FUNCTION_BLOCK FB_Janitza
VAR_IN_OUT
	get					: ST_PowerMonitor_get;
END_VAR
VAR
	MBRead: FB_MBReadRegs;
	w_MBStartAddress	:	WORD;
	//Set 1 is bigger, as this includes voltage measurements.
	DataBuffer		: 	ARRAY[0..62] OF REAL;
	SecondDataBuffer		: 	ARRAY[0..62] OF REAL;
	tempword	:	dword;	
	temp	:	BOOL;
	UI_Iterator	:	UINT;
	//retrieve new data every 100ms
	GetDataTimer	:	TON := (PT := TIME#100MS);
END_VAR

VAR_INPUT
	ReadData: BOOL;
	b_TNmodeEnable		AT %Q* : BOOL;
END_VAR

VAR
	ast_InputPowerlockData	:	ARRAY[1..2] OF ST_Powerlockdata;
	ast_OutputPowerlockData	:	ARRAY[1..3] OF ST_Powerlockdata;

	StartTransmissionEdge : R_Trig;
	TransmissionDone	:	F_trig;
	
	ui_MBRetryCount	:	uint;
	
	b_busy: BOOL;
	b_CommError: BOOL;
	udi_errid: UDINT;
	udi_cbread: UDINT;
	
	testWord	:	DWORD;
	testWordB	:	WORD;
	testWordC	:	WORD;
END_VAR



//While ReadData is true, initiate data transfer every 100ms;
GetDataTimer(in:= ((NOT GetDataTimer.Q) AND ReadData));

//ReadJanitzaData();
ReadDataSFC();

ACTION aCombineInputData:
IF PowerMeterConfig.b_InputFieldsAvailable THEN
	//Combine shared data from output fields into get struct
	get.InputField.r_Current[Phases.L1] :=	get.InputField.ar_PowerlockCurrents[1][Phases.L1] + 
											get.InputField.ar_PowerlockCurrents[2][Phases.L1];
	
	get.InputField.r_Current[Phases.L2] :=	get.InputField.ar_PowerlockCurrents[1][Phases.L2] + 
											get.InputField.ar_PowerlockCurrents[2][Phases.L2];
	
	get.InputField.r_Current[Phases.L3] :=	get.InputField.ar_PowerlockCurrents[1][Phases.L3] + 
											get.InputField.ar_PowerlockCurrents[2][Phases.L3];			
	
	get.InputField.r_Current[Phases.N] :=	get.InputField.ar_PowerlockCurrents[1][Phases.N] + 
											get.InputField.ar_PowerlockCurrents[2][Phases.N];			
	
	get.InputField.r_Current[Phases.AVG] :=	(get.InputField.r_Current[Phases.L1] + 
											get.InputField.r_Current[Phases.L2] +
											get.InputField.r_Current[Phases.L3])/3;							
	
	Get.InputField.r_ActivePhasePower[Phases.L1]	:=	ast_InputPowerLockData[1].r_ActivePhasePower[Phases.L1] + 
														ast_InputPowerLockData[2].r_ActivePhasePower[Phases.L1];
	
	Get.InputField.r_ActivePhasePower[Phases.L2]	:=	ast_InputPowerLockData[1].r_ActivePhasePower[Phases.L2] + 
														ast_InputPowerLockData[2].r_ActivePhasePower[Phases.L2];
														
	Get.InputField.r_ActivePhasePower[Phases.L3]	:=	ast_InputPowerLockData[1].r_ActivePhasePower[Phases.L3] + 
														ast_InputPowerLockData[2].r_ActivePhasePower[Phases.L3];
														
	Get.InputField.r_ActivePhasePower[Phases.AVG]	:=	ast_InputPowerLockData[1].r_ActivePhasePower[Phases.AVG] + 
														ast_InputPowerLockData[2].r_ActivePhasePower[Phases.AVG];									
	
														
														
	Get.InputField.r_ApparentPhasePower[Phases.L1]	:=	ast_InputPowerLockData[1].r_ApparentPhasePower[Phases.L1] + 
														ast_InputPowerLockData[2].r_ApparentPhasePower[Phases.L1];
	
	Get.InputField.r_ApparentPhasePower[Phases.L2]	:=	ast_InputPowerLockData[1].r_ApparentPhasePower[Phases.L2] + 
														ast_InputPowerLockData[2].r_ApparentPhasePower[Phases.L2];
														
	Get.InputField.r_ApparentPhasePower[Phases.L3]	:=	ast_InputPowerLockData[1].r_ApparentPhasePower[Phases.L3] + 
														ast_InputPowerLockData[2].r_ApparentPhasePower[Phases.L3];
														
	Get.InputField.r_ApparentPhasePower[Phases.AVG]	:=	ast_InputPowerLockData[1].r_ApparentPhasePower[Phases.AVG] + 
														ast_InputPowerLockData[2].r_ApparentPhasePower[Phases.AVG];	

														
														
	Get.InputField.r_ReactivePhasePower[Phases.L1]	:=	ast_InputPowerLockData[1].r_ReactivePhasePower[Phases.L1] + 
														ast_InputPowerLockData[2].r_ReactivePhasePower[Phases.L1];
	
	Get.InputField.r_ReactivePhasePower[Phases.L2]	:=	ast_InputPowerLockData[1].r_ReactivePhasePower[Phases.L2] + 
														ast_InputPowerLockData[2].r_ReactivePhasePower[Phases.L2];
														
	Get.InputField.r_ReactivePhasePower[Phases.L3]	:=	ast_InputPowerLockData[1].r_ReactivePhasePower[Phases.L3] + 
														ast_InputPowerLockData[2].r_ReactivePhasePower[Phases.L3];
														
	Get.InputField.r_ReactivePhasePower[Phases.AVG]	:=	ast_InputPowerLockData[1].r_ReactivePhasePower[Phases.AVG] + 
														ast_InputPowerLockData[2].r_ReactivePhasePower[Phases.AVG];	


										
	Get.InputField.r_ActivePower		:=	ast_InputPowerLockData[1].r_ActivePower + 
											ast_InputPowerLockData[2].r_ActivePower;
	
	Get.InputField.r_ApparentPower		:=	ast_InputPowerLockData[1].r_ApparentPower + 
											ast_InputPowerLockData[2].r_ApparentPower;
											
	Get.InputField.r_ReactivePower		:=	ast_InputPowerLockData[1].r_ReactivePower + 
											ast_InputPowerLockData[2].r_ReactivePower;
	
	Get.InputField.r_EnergyConsumed		:=	ast_InputPowerLockData[1].r_EnergyConsumed + 
											ast_InputPowerLockData[2].r_EnergyConsumed;
	
	Get.InputField.r_EnergySupplied		:=	ast_InputPowerLockData[1].r_EnergySupplied + 
											ast_InputPowerLockData[2].r_EnergySupplied;
	
	get.InputField.r_PowerFactor[Phases.L1] :=		(ast_InputPowerLockData[1].ar_PowerFactor[Phases.L1] + 
													ast_InputPowerLockData[2].ar_PowerFactor[Phases.L1] )/2;	
														
	get.InputField.r_PowerFactor[Phases.L2] :=		(ast_InputPowerLockData[1].ar_PowerFactor[Phases.L2] + 
													ast_InputPowerLockData[2].ar_PowerFactor[Phases.L2])/2;		
	
	get.InputField.r_PowerFactor[Phases.L3] :=		(ast_InputPowerLockData[1].ar_PowerFactor[Phases.L3] + 
													ast_InputPowerLockData[2].ar_PowerFactor[Phases.L3])/2;
	
	get.InputField.r_THD[Phases.L1] 		:=		(ast_InputPowerLockData[1].ar_THD[Phases.L1] + 
													ast_InputPowerLockData[2].ar_THD[Phases.L1])/2;
														
	get.InputField.r_THD[Phases.L2] 		:=		(ast_InputPowerLockData[1].ar_THD[Phases.L2] + 
													ast_InputPowerLockData[2].ar_THD[Phases.L2])/2;	
	
	get.InputField.r_THD[Phases.L3]		 	:=		(ast_InputPowerLockData[1].ar_THD[Phases.L3] + 
													ast_InputPowerLockData[2].ar_THD[Phases.L3])/2;											
	
	get.InputField.r_PowerFactor[Phases.AVG] :=	(get.InputField.r_PowerFactor[Phases.L1] + 
													get.InputField.r_PowerFactor[Phases.L2] + 
													get.InputField.r_PowerFactor[Phases.L3])/3;		
	
	get.InputField.r_THD[Phases.AVG] :=			(get.InputField.r_THD[Phases.L1] + 
													get.InputField.r_THD[Phases.L2] + 
													get.InputField.r_THD[Phases.L3])/3;
end_if
END_ACTION

ACTION aCombineOutputData:

//Combine shared data from output fields into get struct
get.OutputField.r_Current[Phases.L1] :=	get.OutputField.ar_PowerlockCurrents[1][Phases.L1] + 
										get.OutputField.ar_PowerlockCurrents[2][Phases.L1] + 
										get.OutputField.ar_PowerlockCurrents[3][Phases.L1];

get.OutputField.r_Current[Phases.L2] :=	get.OutputField.ar_PowerlockCurrents[1][Phases.L2] + 
										get.OutputField.ar_PowerlockCurrents[2][Phases.L2] + 
										get.OutputField.ar_PowerlockCurrents[3][Phases.L2];

get.OutputField.r_Current[Phases.L3] :=	get.OutputField.ar_PowerlockCurrents[1][Phases.L3] + 
										get.OutputField.ar_PowerlockCurrents[2][Phases.L3] + 
										get.OutputField.ar_PowerlockCurrents[3][Phases.L3];			

get.OutputField.r_Current[Phases.N] :=	get.OutputField.ar_PowerlockCurrents[1][Phases.N] + 
										get.OutputField.ar_PowerlockCurrents[2][Phases.N] + 
										get.OutputField.ar_PowerlockCurrents[3][Phases.N];			

get.OutputField.r_Current[Phases.AVG] :=	(get.OutputField.r_Current[Phases.L1] + 
											get.OutputField.r_Current[Phases.L2] +
											get.OutputField.r_Current[Phases.L3])/3;							

Get.OutputField.r_ActivePhasePower[Phases.L1]	:=	ast_OutputPowerLockData[1].r_ActivePhasePower[Phases.L1] + 
													ast_OutputPowerLockData[2].r_ActivePhasePower[Phases.L1] +
													ast_OutputPowerLockData[3].r_ActivePhasePower[Phases.L1];
	
Get.OutputField.r_ActivePhasePower[Phases.L2]	:=	ast_OutputPowerLockData[1].r_ActivePhasePower[Phases.L2] + 
													ast_OutputPowerLockData[2].r_ActivePhasePower[Phases.L2] +
													ast_OutputPowerLockData[3].r_ActivePhasePower[Phases.L2];
														
Get.OutputField.r_ActivePhasePower[Phases.L3]	:=	ast_OutputPowerLockData[1].r_ActivePhasePower[Phases.L3] + 
													ast_OutputPowerLockData[2].r_ActivePhasePower[Phases.L3] + 
													ast_OutputPowerLockData[3].r_ActivePhasePower[Phases.L3];
														
Get.OutputField.r_ActivePhasePower[Phases.AVG]	:=	ast_OutputPowerLockData[1].r_ActivePhasePower[Phases.AVG] + 
													ast_OutputPowerLockData[2].r_ActivePhasePower[Phases.AVG] +
													ast_OutputPowerLockData[3].r_ActivePhasePower[Phases.AVG];									
	
														
														
Get.OutputField.r_ApparentPhasePower[Phases.L1]	:=	ast_OutputPowerLockData[1].r_ApparentPhasePower[Phases.L1] + 
													ast_OutputPowerLockData[2].r_ApparentPhasePower[Phases.L1] +
													ast_OutputPowerLockData[3].r_ApparentPhasePower[Phases.L1];
	
Get.OutputField.r_ApparentPhasePower[Phases.L2]	:=	ast_OutputPowerLockData[1].r_ApparentPhasePower[Phases.L2] + 
													ast_OutputPowerLockData[2].r_ApparentPhasePower[Phases.L2] +
													ast_OutputPowerLockData[3].r_ApparentPhasePower[Phases.L2];
														
Get.OutputField.r_ApparentPhasePower[Phases.L3]	:=	ast_OutputPowerLockData[1].r_ApparentPhasePower[Phases.L3] + 
													ast_OutputPowerLockData[2].r_ApparentPhasePower[Phases.L3] +
													ast_OutputPowerLockData[3].r_ApparentPhasePower[Phases.L3];
														
Get.OutputField.r_ApparentPhasePower[Phases.AVG]:=	ast_OutputPowerLockData[1].r_ApparentPhasePower[Phases.AVG] + 
													ast_OutputPowerLockData[2].r_ApparentPhasePower[Phases.AVG] +
													ast_OutputPowerLockData[3].r_ApparentPhasePower[Phases.AVG];	
														
													
													
Get.OutputField.r_ReactivePhasePower[Phases.L1]	:=	ast_OutputPowerLockData[1].r_ReactivePhasePower[Phases.L1] + 
													ast_OutputPowerLockData[2].r_ReactivePhasePower[Phases.L1] +
													ast_OutputPowerLockData[3].r_ReactivePhasePower[Phases.L1];	
	
Get.OutputField.r_ReactivePhasePower[Phases.L2]	:=	ast_OutputPowerLockData[1].r_ReactivePhasePower[Phases.L2] + 
													ast_OutputPowerLockData[2].r_ReactivePhasePower[Phases.L2] +
													ast_OutputPowerLockData[3].r_ReactivePhasePower[Phases.L2];	
														
Get.OutputField.r_ReactivePhasePower[Phases.L3]	:=	ast_OutputPowerLockData[1].r_ReactivePhasePower[Phases.L3] + 
													ast_OutputPowerLockData[2].r_ReactivePhasePower[Phases.L3] +
													ast_OutputPowerLockData[3].r_ReactivePhasePower[Phases.L3];	
														
Get.OutputField.r_ReactivePhasePower[Phases.AVG]:=	ast_OutputPowerLockData[1].r_ReactivePhasePower[Phases.AVG] + 
													ast_OutputPowerLockData[2].r_ReactivePhasePower[Phases.AVG] +	
													ast_OutputPowerLockData[3].r_ReactivePhasePower[Phases.AVG];												
											
											
Get.OutputField.r_ActivePower		:=	ast_OutputPowerLockData[1].r_ActivePower + 
										ast_OutputPowerLockData[2].r_ActivePower + 
										ast_OutputPowerLockData[3].r_ActivePower;

Get.OutputField.r_ApparentPower		:=	ast_OutputPowerLockData[1].r_ApparentPower + 
										ast_OutputPowerLockData[2].r_ApparentPower + 
										ast_OutputPowerLockData[3].r_ApparentPower;

Get.OutputField.r_ReactivePower		:=	ast_OutputPowerLockData[1].r_ReactivePower + 
										ast_OutputPowerLockData[2].r_ReactivePower + 
										ast_OutputPowerLockData[3].r_ReactivePower;

Get.OutputField.r_EnergyConsumed	:=	ast_OutputPowerLockData[1].r_EnergyConsumed + 
										ast_OutputPowerLockData[2].r_EnergyConsumed + 
										ast_OutputPowerLockData[3].r_EnergyConsumed;

Get.OutputField.r_EnergySupplied	:=	ast_OutputPowerLockData[1].r_EnergySupplied + 
										ast_OutputPowerLockData[2].r_EnergySupplied + 
										ast_OutputPowerLockData[3].r_EnergySupplied;

//if 3 output fields are available, calculate averages over 3 fields. Otherwise over 2
IF PowerMeterConfig.b_ThirdOutputFieldAvailable THEN
	get.OutputField.r_PowerFactor[Phases.L1] :=		(ast_OutputPowerLockData[1].ar_PowerFactor[Phases.L1] + 
													ast_OutputPowerLockData[2].ar_PowerFactor[Phases.L1] + 
													ast_OutputPowerLockData[3].ar_PowerFactor[Phases.L1])/3;	
													
	get.OutputField.r_PowerFactor[Phases.L2] :=		(ast_OutputPowerLockData[1].ar_PowerFactor[Phases.L2] + 
													ast_OutputPowerLockData[2].ar_PowerFactor[Phases.L2] + 
													ast_OutputPowerLockData[3].ar_PowerFactor[Phases.L2])/3;		

	get.OutputField.r_PowerFactor[Phases.L3] :=		(ast_OutputPowerLockData[1].ar_PowerFactor[Phases.L3] + 
													ast_OutputPowerLockData[2].ar_PowerFactor[Phases.L3] + 
													ast_OutputPowerLockData[3].ar_PowerFactor[Phases.L3])/3;	

	get.OutputField.r_THD[Phases.L1] 		:=		(ast_OutputPowerLockData[1].ar_THD[Phases.L1] + 
													ast_OutputPowerLockData[2].ar_THD[Phases.L1] + 
													ast_OutputPowerLockData[3].ar_THD[Phases.L1])/3;	
													
	get.OutputField.r_THD[Phases.L2] 		:=		(ast_OutputPowerLockData[1].ar_THD[Phases.L2] + 
													ast_OutputPowerLockData[2].ar_THD[Phases.L2] + 
													ast_OutputPowerLockData[3].ar_THD[Phases.L2])/3;		

	get.OutputField.r_THD[Phases.L3]		 :=		(ast_OutputPowerLockData[1].ar_THD[Phases.L3] + 
													ast_OutputPowerLockData[2].ar_THD[Phases.L3] + 
													ast_OutputPowerLockData[3].ar_THD[Phases.L3])/3;														
ELSE
	get.OutputField.r_PowerFactor[Phases.L1] :=		(ast_OutputPowerLockData[1].ar_PowerFactor[Phases.L1] + 
													ast_OutputPowerLockData[2].ar_PowerFactor[Phases.L1] )/2;	
													
	get.OutputField.r_PowerFactor[Phases.L2] :=		(ast_OutputPowerLockData[1].ar_PowerFactor[Phases.L2] + 
													ast_OutputPowerLockData[2].ar_PowerFactor[Phases.L2])/2;		

	get.OutputField.r_PowerFactor[Phases.L3] :=		(ast_OutputPowerLockData[1].ar_PowerFactor[Phases.L3] + 
													ast_OutputPowerLockData[2].ar_PowerFactor[Phases.L3])/2;

	get.OutputField.r_THD[Phases.L1] 		:=		(ast_OutputPowerLockData[1].ar_THD[Phases.L1] + 
													ast_OutputPowerLockData[2].ar_THD[Phases.L1])/2;
													
	get.OutputField.r_THD[Phases.L2] 		:=		(ast_OutputPowerLockData[1].ar_THD[Phases.L2] + 
													ast_OutputPowerLockData[2].ar_THD[Phases.L2])/2;	

	get.OutputField.r_THD[Phases.L3]		 :=		(ast_OutputPowerLockData[1].ar_THD[Phases.L3] + 
													ast_OutputPowerLockData[2].ar_THD[Phases.L3])/2;											
END_IF



get.OutputField.r_PowerFactor[Phases.AVG] :=	(get.OutputField.r_PowerFactor[Phases.L1] + 
												get.OutputField.r_PowerFactor[Phases.L2] + 
												get.OutputField.r_PowerFactor[Phases.L3])/3;		

get.OutputField.r_THD[Phases.AVG] :=			(get.OutputField.r_THD[Phases.L1] + 
												get.OutputField.r_THD[Phases.L2] + 
												get.OutputField.r_THD[Phases.L3])/3;
END_ACTION

ACTION aReadInputField1:

IF NOT PowerMeterConfig.b_InputFieldsAvailable THEN
	//skip this step if input fields are not in use
	SFCTip := TRUE;
ELSE
	
	IF PowerMeterconfig.b_ThirdOutputFieldAvailable THEN
		//if third output field is available, Input field is connected to module 2, so inputfield 1 is address 19600
		w_MBStartAddress := 19600;
	ELSE
		//if no third output field is available, Input field is connected to module 1, so inputfield 1 is address 19400
		w_MBStartAddress := 19400;
	END_IF

	MBRead(
	sIPAddr := PowerMeterConfig.IP_JANITZA,
	nTCPPort := PowerMeterConfig.MBPort_Janitza,
	nUnitID := 1,//16#FF;
	nMBAddr := w_MBStartAddress,
	nQuantity := 50*2,
	cbLength := SIZEOF(DataBuffer),
	pDestAddr := ADR(DataBuffer),
	bExecute := NOT (b_busy OR TransmissionDone.Q),	//	<- werkt dit niet gewoon?
	bBusy => b_busy,
	bError => b_CommError,
	nErrId => udi_errid,
	cbRead => udi_cbread,
	tTimeout := T#25MS
	);
	
	TransmissionDone(clk := b_busy);
	
	IF TransmissionDone.q THEN
		IF NOT b_CommError  THEN	
			
			FOR UI_Iterator := 0 TO 50 BY 1 DO
				DataBuffer[UI_Iterator] := ChangeRealEndianess(DataBuffer[UI_Iterator]);
			END_FOR 
			//field specific data, keep separate at first. Then combine data into get struct in a later step.
			get.InputField.ar_PowerlockCurrents[1][Phases.L1] := DataBuffer[0];
			get.InputField.ar_PowerlockCurrents[1][Phases.L2] := DataBuffer[1];
			get.InputField.ar_PowerlockCurrents[1][Phases.L3] := DataBuffer[2];
			get.InputField.ar_PowerlockCurrents[1][Phases.N] := DataBuffer[3];
			
			ast_InputPowerLockData[1].r_ActivePhasePower[phases.L1] := DataBuffer[4];
       		ast_InputPowerLockData[1].r_ActivePhasePower[phases.L2] := DataBuffer[5];
			ast_InputPowerLockData[1].r_ActivePhasePower[phases.L3] := DataBuffer[6];
			ast_InputPowerLockData[1].r_ActivePhasePower[phases.AVG] := (DataBuffer[4] + DataBuffer[5] + DataBuffer[6])/3;
		    
			ast_InputPowerLockData[1].r_ApparentPhasePower[phases.L1] := DataBuffer[8];
       		ast_InputPowerLockData[1].r_ApparentPhasePower[phases.L2] := DataBuffer[9];
			ast_InputPowerLockData[1].r_ApparentPhasePower[phases.L3] := DataBuffer[10];
			ast_InputPowerLockData[1].r_ApparentPhasePower[phases.AVG] := (DataBuffer[8] + DataBuffer[9] + DataBuffer[10])/3;
		    
			ast_InputPowerLockData[1].r_ReactivePhasePower[phases.L1] := DataBuffer[12];
       		ast_InputPowerLockData[1].r_ReactivePhasePower[phases.L2] := DataBuffer[13];
			ast_InputPowerLockData[1].r_ReactivePhasePower[phases.L3] := DataBuffer[14];
			ast_InputPowerLockData[1].r_ReactivePhasePower[phases.AVG] := (DataBuffer[12] + DataBuffer[13] + DataBuffer[14])/3;
		    
			ast_InputPowerLockData[1].r_ActivePower := DataBuffer[7];
			ast_InputPowerLockData[1].r_ApparentPower := DataBuffer[11];
			ast_InputPowerLockData[1].r_ReactivePower := DataBuffer[15];
					               
			ast_InputPowerLockData[1].ar_PowerFactor[Phases.L1] := DataBuffer[16];
			ast_InputPowerLockData[1].ar_PowerFactor[Phases.L2] := DataBuffer[17];
			ast_InputPowerLockData[1].ar_PowerFactor[Phases.L3] := DataBuffer[18];
			ast_InputPowerLockData[1].ar_PowerFactor[Phases.AVG] := (DataBuffer[16] + DataBuffer[17] + DataBuffer[18])/3;
					               
			ast_InputPowerLockData[1].r_EnergyConsumed	:=  DataBuffer[26];
			ast_InputPowerLockData[1].r_EnergySupplied 	:=	DataBuffer[30];
					               
			ast_InputPowerLockData[1].ar_THD[Phases.L1] := DataBuffer[47];
			ast_InputPowerLockData[1].ar_THD[Phases.L2] := DataBuffer[48];
			ast_InputPowerLockData[1].ar_THD[Phases.L3] := DataBuffer[49];
				
			ui_MBRetryCount := 0;
			sfctip := TRUE;
		ELSE
			ui_MBRetryCount := ui_MBRetryCount + 1;
			
			IF ui_MBRetryCount > 1 THEN
				get.events.b_MBCommWarning := TRUE;
			END_IF	
			
			//if comm fails 5 times in a row. try next input
			IF ui_MBRetryCount > 4 THEN
				get.Events.b_MBCommError := TRUE;
				sfctip := TRUE;
			END_IF
		END_IF
	END_IF
END_IF
END_ACTION

ACTION aReadInputField2:

IF NOT PowerMeterConfig.b_InputFieldsAvailable THEN
	//skip this step if input fields are not in use
	SFCTip := TRUE;
ELSE
	
	IF PowerMeterconfig.b_ThirdOutputFieldAvailable THEN
		//if third output field is available, Input field is connected to module 2, so inputfield 2 is address 19700
		w_MBStartAddress := 19700;
	ELSE
		//if no third output field is available, Input field is connected to module 1, so inputfield 2 is address 19500
		w_MBStartAddress := 19500;
	END_IF

	MBRead(
	sIPAddr := PowerMeterConfig.IP_JANITZA,
	nTCPPort := PowerMeterConfig.MBPort_Janitza,
	nUnitID := 1,//16#FF;
	nMBAddr := w_MBStartAddress,
	nQuantity := 50*2,
	cbLength := SIZEOF(DataBuffer),
	pDestAddr := ADR(DataBuffer),
	bExecute := NOT (b_busy OR TransmissionDone.Q),	//	<- werkt dit niet gewoon?
	bBusy => b_busy,
	bError => b_CommError,
	nErrId => udi_errid,
	cbRead => udi_cbread,
	tTimeout := T#25MS
	);
	
	TransmissionDone(clk := b_busy);
	
	IF TransmissionDone.q THEN
		IF NOT b_CommError THEN	
			
			FOR UI_Iterator := 0 TO 50 BY 1 DO
				DataBuffer[UI_Iterator] := ChangeRealEndianess(DataBuffer[UI_Iterator]);
			END_FOR 
			
			//field specific data, keep separate at first. Then combine data into get struct in a later step.
			get.InputField.ar_PowerlockCurrents[2][Phases.L1] := DataBuffer[0];
			get.InputField.ar_PowerlockCurrents[2][Phases.L2] := DataBuffer[1];
			get.InputField.ar_PowerlockCurrents[2][Phases.L3] := DataBuffer[2];
			get.InputField.ar_PowerlockCurrents[2][Phases.N] := DataBuffer[3];
			
			ast_InputPowerLockData[2].r_ActivePhasePower[phases.L1] := DataBuffer[4];
       		ast_InputPowerLockData[2].r_ActivePhasePower[phases.L2] := DataBuffer[5];
			ast_InputPowerLockData[2].r_ActivePhasePower[phases.L3] := DataBuffer[6];
			ast_InputPowerLockData[2].r_ActivePhasePower[phases.AVG] := (DataBuffer[4] + DataBuffer[5] + DataBuffer[6])/3;
		                           
			ast_InputPowerLockData[2].r_ApparentPhasePower[phases.L1] := DataBuffer[8];
       		ast_InputPowerLockData[2].r_ApparentPhasePower[phases.L2] := DataBuffer[9];
			ast_InputPowerLockData[2].r_ApparentPhasePower[phases.L3] := DataBuffer[10];
			ast_InputPowerLockData[2].r_ApparentPhasePower[phases.AVG] := (DataBuffer[8] + DataBuffer[9] + DataBuffer[10])/3;
		                           
			ast_InputPowerLockData[2].r_ReactivePhasePower[phases.L1] := DataBuffer[12];
       		ast_InputPowerLockData[2].r_ReactivePhasePower[phases.L2] := DataBuffer[13];
			ast_InputPowerLockData[2].r_ReactivePhasePower[phases.L3] := DataBuffer[14];
			ast_InputPowerLockData[2].r_ReactivePhasePower[phases.AVG] := (DataBuffer[12] + DataBuffer[13] + DataBuffer[14])/3;
		    			
			ast_InputPowerLockData[2].r_ActivePower := DataBuffer[7];
			ast_InputPowerLockData[2].r_ApparentPower := DataBuffer[11];
			ast_InputPowerLockData[2].r_ReactivePower := DataBuffer[15];
					               
			ast_InputPowerLockData[2].ar_PowerFactor[Phases.L1] := DataBuffer[16];
			ast_InputPowerLockData[2].ar_PowerFactor[Phases.L2] := DataBuffer[17];
			ast_InputPowerLockData[2].ar_PowerFactor[Phases.L3] := DataBuffer[18];
			ast_InputPowerLockData[2].ar_PowerFactor[Phases.AVG] := (DataBuffer[16] + DataBuffer[17] + DataBuffer[18])/3;
					               
			ast_InputPowerLockData[2].r_EnergyConsumed	:=  DataBuffer[26];
			ast_InputPowerLockData[2].r_EnergySupplied 	:=	DataBuffer[30];
					               
			ast_InputPowerLockData[2].ar_THD[Phases.L1] := DataBuffer[47];
			ast_InputPowerLockData[2].ar_THD[Phases.L2] := DataBuffer[48];
			ast_InputPowerLockData[2].ar_THD[Phases.L3] := DataBuffer[49];
				
			ui_MBRetryCount := 0;
			sfctip := TRUE;
		ELSE
			ui_MBRetryCount := ui_MBRetryCount + 1;
			
			
			IF ui_MBRetryCount > 1 THEN
				get.events.b_MBCommWarning := TRUE;
			END_IF	
			
			//if comm fails 5 times in a row. try next input
			IF ui_MBRetryCount > 4 THEN
				get.Events.b_MBCommError := TRUE;
				sfctip := TRUE;
			END_IF
		END_IF
	END_IF
END_IF
END_ACTION

ACTION aReadInternalField:

MBRead(
sIPAddr := PowerMeterConfig.IP_JANITZA,
nTCPPort := PowerMeterConfig.MBPort_Janitza,
nUnitID := 1,//16#FF;
nMBAddr := 19300,
nQuantity := 50*2,
cbLength := SIZEOF(DataBuffer),
pDestAddr := ADR(DataBuffer),
bExecute := NOT (b_busy OR TransmissionDone.Q),	//	<- werkt dit niet gewoon?
bBusy => b_busy,
bError => b_CommError,
nErrId => udi_errid,
cbRead => udi_cbread,
tTimeout := T#25MS
);

TransmissionDone(clk := b_busy);

IF TransmissionDone.q THEN
	IF NOT b_CommError  THEN	
		
		FOR UI_Iterator := 0 TO 50 BY 1 DO
			DataBuffer[UI_Iterator] := ChangeRealEndianess(DataBuffer[UI_Iterator]);
		END_FOR 
		
		//field specific data, keep separate at first. Then combine data into get struct in a later step.
		get.InternalSupply.r_Current[Phases.L1] := DataBuffer[0];
		get.InternalSupply.r_Current[Phases.L2] := DataBuffer[1];
		get.InternalSupply.r_Current[Phases.L3] := DataBuffer[2];
		get.InternalSupply.r_Current[Phases.N] := DataBuffer[3];
		get.InternalSupply.r_Current[Phases.AVG] := (DataBuffer[0] + DataBuffer[1] + DataBuffer[2])/3;
		
		get.InternalSupply.r_ActivePhasePower[phases.L1] := DataBuffer[4];
   		get.InternalSupply.r_ActivePhasePower[phases.L2] := DataBuffer[5];
		get.InternalSupply.r_ActivePhasePower[phases.L3] := DataBuffer[6];
		get.InternalSupply.r_ActivePhasePower[phases.AVG] := (DataBuffer[4] + DataBuffer[5] + DataBuffer[6])/3;
		
		get.InternalSupply.r_ApparentPhasePower[phases.L1] := DataBuffer[8];
   		get.InternalSupply.r_ApparentPhasePower[phases.L2] := DataBuffer[9];
		get.InternalSupply.r_ApparentPhasePower[phases.L3] := DataBuffer[10];
		get.InternalSupply.r_ApparentPhasePower[phases.AVG] := (DataBuffer[8] + DataBuffer[9] + DataBuffer[10])/3;
		
		get.InternalSupply.r_ReactivePhasePower[phases.L1] := DataBuffer[12];
   		get.InternalSupply.r_ReactivePhasePower[phases.L2] := DataBuffer[13];
		get.InternalSupply.r_ReactivePhasePower[phases.L3] := DataBuffer[14];
		get.InternalSupply.r_ReactivePhasePower[phases.AVG] := (DataBuffer[12] + DataBuffer[13] + DataBuffer[14])/3;
		    				                        
		get.InternalSupply.r_ActivePower := DataBuffer[7];
		get.InternalSupply.r_ApparentPower := DataBuffer[11];
		get.InternalSupply.r_ReactivePower := DataBuffer[15];
        
		get.InternalSupply.r_PowerFactor[Phases.L1] := DataBuffer[16];
		get.InternalSupply.r_PowerFactor[Phases.L2] := DataBuffer[17];
		get.InternalSupply.r_PowerFactor[Phases.L3] := DataBuffer[18];
		get.InternalSupply.r_PowerFactor[Phases.AVG] := (DataBuffer[16] + DataBuffer[17] + DataBuffer[18])/3;
		
		get.InternalSupply.r_EnergyConsumed	:=  DataBuffer[26];
		get.InternalSupply.r_EnergySupplied 	:=	DataBuffer[30];
		
		get.InternalSupply.r_THD[Phases.L1] := DataBuffer[47];
		get.InternalSupply.r_THD[Phases.L2] := DataBuffer[48];
		get.InternalSupply.r_THD[Phases.L3] := DataBuffer[49];
			
		ui_MBRetryCount := 0;
		sfctip := TRUE;
	ELSE
		ui_MBRetryCount := ui_MBRetryCount + 1;
				
		IF ui_MBRetryCount > 1 THEN
			get.events.b_MBCommWarning := TRUE;
		END_IF	
		
		//if comm fails 5 times in a row. try next input
		IF ui_MBRetryCount > 4 THEN
			get.Events.b_MBCommError := TRUE;
			sfctip := TRUE;
		END_IF
	END_IF
END_IF
END_ACTION

ACTION aReadOutputField1:

MBRead(
sIPAddr := PowerMeterConfig.IP_JANITZA,
nTCPPort := PowerMeterConfig.MBPort_Janitza,
nUnitID := 1,
nMBAddr := 19000,
nQuantity := 61*2,
cbLength := SIZEOF(DataBuffer),
pDestAddr := ADR(DataBuffer),
bExecute := NOT (b_busy OR TransmissionDone.Q),	//	<- werkt dit niet gewoon?
bBusy => b_busy,
bError => b_CommError,
nErrId => udi_errid,
cbRead => udi_cbread,
tTimeout := T#25MS
);

TransmissionDone(clk := b_busy);

IF TransmissionDone.q THEN
	Temp := FALSE;
	IF NOT b_CommError then
		//General inputfield data, can be pushed to get struct immediately
		
		FOR UI_Iterator := 0 TO 61 BY 1 DO
			DataBuffer[UI_Iterator] := ChangeRealEndianess(DataBuffer[UI_Iterator]);
		END_FOR 
		
		get.OutputField.r_PhaseVoltage[Phases.L1] := DataBuffer[0];
		get.OutputField.r_PhaseVoltage[Phases.L2] := DataBuffer[1];
		get.OutputField.r_PhaseVoltage[Phases.L3] := DataBuffer[2];
		get.OutputField.r_PhaseVoltage[Phases.AVG] := (DataBuffer[0]+DataBuffer[1]+DataBuffer[2])/3;
		
		get.OutputField.r_LineVoltage[Phases.L1] := DataBuffer[3];
		get.OutputField.r_LineVoltage[Phases.L2] := DataBuffer[4];
		get.OutputField.r_LineVoltage[Phases.L3] := DataBuffer[5];
		get.OutputField.r_LineVoltage[Phases.AVG] := (DataBuffer[3]+DataBuffer[4]+DataBuffer[5])/3;
		
		get.OutputField.r_Frequency	:= DataBuffer[25];
		
		CASE REAL_TO_INT(DataBuffer[26]) OF
			-1 	:	get.OutputField.e_ACrotationStatus := eACRotationState.Left;
			1	:	get.OutputField.e_ACrotationStatus := eACRotationState.Right;
			0	:	get.OutputField.e_ACrotationStatus := eACRotationState.None;
		END_CASE

		//field specific data, keep separate at first. Then combine data into get struct in a later step.
		get.OutputField.ar_PowerlockCurrents[1][Phases.L1] := DataBuffer[6];
		get.OutputField.ar_PowerlockCurrents[1][Phases.L2] := DataBuffer[7];
		get.OutputField.ar_PowerlockCurrents[1][Phases.L3] := DataBuffer[8];
		get.OutputField.ar_PowerlockCurrents[1][Phases.N] := DataBuffer[9];
		
		ast_OutputPowerLockData[1].r_ActivePhasePower[phases.L1] := DataBuffer[10];
   		ast_OutputPowerLockData[1].r_ActivePhasePower[phases.L2] := DataBuffer[11];
		ast_OutputPowerLockData[1].r_ActivePhasePower[phases.L3] := DataBuffer[12];
		ast_OutputPowerLockData[1].r_ActivePhasePower[phases.AVG] := (DataBuffer[10] + DataBuffer[11] + DataBuffer[12])/3;
		                        
		ast_OutputPowerLockData[1].r_ApparentPhasePower[phases.L1] := DataBuffer[14];
   		ast_OutputPowerLockData[1].r_ApparentPhasePower[phases.L2] := DataBuffer[15];
		ast_OutputPowerLockData[1].r_ApparentPhasePower[phases.L3] := DataBuffer[16];
		ast_OutputPowerLockData[1].r_ApparentPhasePower[phases.AVG] := (DataBuffer[14] + DataBuffer[15] + DataBuffer[16])/3;
		                        
		ast_OutputPowerLockData[1].r_ReactivePhasePower[phases.L1] := DataBuffer[18];
   		ast_OutputPowerLockData[1].r_ReactivePhasePower[phases.L2] := DataBuffer[19];
		ast_OutputPowerLockData[1].r_ReactivePhasePower[phases.L3] := DataBuffer[20];
		ast_OutputPowerLockData[1].r_ReactivePhasePower[phases.AVG] := (DataBuffer[18] + DataBuffer[19] + DataBuffer[20])/3;
		    				                        
		ast_OutputPowerLockData[1].r_ActivePower := DataBuffer[13];
		ast_OutputPowerLockData[1].r_ApparentPower := DataBuffer[17];
		ast_OutputPowerLockData[1].r_ReactivePower := DataBuffer[21];

		ast_OutputPowerLockData[1].ar_PowerFactor[Phases.L1] := DataBuffer[22];
		ast_OutputPowerLockData[1].ar_PowerFactor[Phases.L2] := DataBuffer[23];
		ast_OutputPowerLockData[1].ar_PowerFactor[Phases.L3] := DataBuffer[24];
		ast_OutputPowerLockData[1].ar_PowerFactor[Phases.AVG] := (DataBuffer[22] + DataBuffer[23] + DataBuffer[24])/3;
		
		ast_OutputPowerLockData[1].r_EnergyConsumed	:=  DataBuffer[34];
		ast_OutputPowerLockData[1].r_EnergySupplied 	:=	DataBuffer[38];

		ast_OutputPowerLockData[1].ar_THD[Phases.L1] := DataBuffer[58];
		ast_OutputPowerLockData[1].ar_THD[Phases.L2] := DataBuffer[59];
		ast_OutputPowerLockData[1].ar_THD[Phases.L3] := DataBuffer[60];
			
		ui_MBRetryCount := 0;
		sfctip := TRUE;
	ELSE
		ui_MBRetryCount := ui_MBRetryCount + 1;
		
		IF ui_MBRetryCount > 1 THEN
			get.events.b_MBCommWarning := TRUE;
		END_IF	
		
		//if comm fails 5 times in a row. try next input
		IF ui_MBRetryCount > 4 THEN
			get.Events.b_MBCommError := TRUE;
			sfctip := TRUE;
		END_IF
	END_IF
END_IF
END_ACTION

ACTION aReadOutputField2:

MBRead(
sIPAddr := PowerMeterConfig.IP_JANITZA,
nTCPPort := PowerMeterConfig.MBPort_Janitza,
nUnitID := 1,//16#FF,
nMBAddr := 19200,
nQuantity := 50*2,
cbLength := SIZEOF(DataBuffer),
pDestAddr := ADR(DataBuffer),
bExecute := NOT (b_busy OR TransmissionDone.Q),	//	<- werkt dit niet gewoon?
bBusy => b_busy,
bError => b_CommError,
nErrId => udi_errid,
cbRead => udi_cbread,
tTimeout := T#25MS
);

TransmissionDone(clk := b_busy);

IF TransmissionDone.q THEN
	IF NOT b_CommError THEN	
		
		FOR UI_Iterator := 0 TO 50 BY 1 DO
			DataBuffer[UI_Iterator] := ChangeRealEndianess(DataBuffer[UI_Iterator]);
		END_FOR 	
	
		get.OutputField.ar_PowerlockCurrents[2][Phases.L1] := DataBuffer[0];
		get.OutputField.ar_PowerlockCurrents[2][Phases.L2] := DataBuffer[1];
		get.OutputField.ar_PowerlockCurrents[2][Phases.L3] := DataBuffer[2];
		get.OutputField.ar_PowerlockCurrents[2][Phases.N] := DataBuffer[3];

		ast_OutputPowerLockData[2].r_ActivePhasePower[phases.L1] := DataBuffer[4];
   		ast_OutputPowerLockData[2].r_ActivePhasePower[phases.L2] := DataBuffer[5];
		ast_OutputPowerLockData[2].r_ActivePhasePower[phases.L3] := DataBuffer[6];
		ast_OutputPowerLockData[2].r_ActivePhasePower[phases.AVG] := (DataBuffer[4] + DataBuffer[5] + DataBuffer[6])/3;
		
		ast_OutputPowerLockData[2].r_ApparentPhasePower[phases.L1] := DataBuffer[8];
   		ast_OutputPowerLockData[2].r_ApparentPhasePower[phases.L2] := DataBuffer[9];
		ast_OutputPowerLockData[2].r_ApparentPhasePower[phases.L3] := DataBuffer[10];
		ast_OutputPowerLockData[2].r_ApparentPhasePower[phases.AVG] := (DataBuffer[8] + DataBuffer[9] + DataBuffer[10])/3;
		
		ast_OutputPowerLockData[2].r_ReactivePhasePower[phases.L1] := DataBuffer[12];
   		ast_OutputPowerLockData[2].r_ReactivePhasePower[phases.L2] := DataBuffer[13];
		ast_OutputPowerLockData[2].r_ReactivePhasePower[phases.L3] := DataBuffer[14];
		ast_OutputPowerLockData[2].r_ReactivePhasePower[phases.AVG] := (DataBuffer[12] + DataBuffer[13] + DataBuffer[14])/3;
		    				                        
		ast_OutputPowerLockData[2].r_ActivePower := DataBuffer[7];
		ast_OutputPowerLockData[2].r_ApparentPower := DataBuffer[11];
		ast_OutputPowerLockData[2].r_ReactivePower := DataBuffer[15];
                                
		ast_OutputPowerLockData[2].ar_PowerFactor[Phases.L1] := DataBuffer[16];
		ast_OutputPowerLockData[2].ar_PowerFactor[Phases.L2] := DataBuffer[17];
		ast_OutputPowerLockData[2].ar_PowerFactor[Phases.L3] := DataBuffer[18];
		ast_OutputPowerLockData[2].ar_PowerFactor[Phases.AVG] := (DataBuffer[16] + DataBuffer[17] + DataBuffer[18])/3;
		                        
		ast_OutputPowerLockData[2].r_EnergyConsumed	:=  DataBuffer[26];
		ast_OutputPowerLockData[2].r_EnergySupplied 	:=	DataBuffer[30];
				                
		ast_OutputPowerLockData[2].ar_THD[Phases.L1] := DataBuffer[47];
		ast_OutputPowerLockData[2].ar_THD[Phases.L2] := DataBuffer[48];
		ast_OutputPowerLockData[2].ar_THD[Phases.L3] := DataBuffer[49];
			
		ui_MBRetryCount := 0;
		sfctip := TRUE;
	ELSE
		ui_MBRetryCount := ui_MBRetryCount + 1;
		
		IF ui_MBRetryCount > 1 THEN
			get.events.b_MBCommWarning := TRUE;
		END_IF	
		
		//if comm fails 5 times in a row. try next input
		IF ui_MBRetryCount > 4 THEN
			get.Events.b_MBCommError := TRUE;
			sfctip := TRUE;
		END_IF
	END_IF
END_IF
END_ACTION

ACTION aReadOutputField3:

IF NOT PowerMeterConfig.b_ThirdOutputFieldAvailable THEN
	//skip this step if third field isn't in use
	SFCTip := TRUE;
ELSE
	MBRead(
	sIPAddr := PowerMeterConfig.IP_JANITZA,
	nTCPPort := PowerMeterConfig.MBPort_Janitza,
	nUnitID := 1,//16#FF;
	nMBAddr := 19400,
	nQuantity := 50*2,
	cbLength := SIZEOF(SecondDataBuffer),
	pDestAddr := ADR(SecondDataBuffer),
	bExecute := NOT (b_busy OR TransmissionDone.Q),	//	<- werkt dit niet gewoon?
	bBusy => b_busy,
	bError => b_CommError,
	nErrId => udi_errid,
	cbRead => udi_cbread,
	tTimeout := T#25MS
	);
	
	TransmissionDone(clk := b_busy);
	
	IF TransmissionDone.q THEN
		IF NOT b_CommError  THEN	
			
			FOR UI_Iterator := 0 TO 50 BY 1 DO
				DataBuffer[UI_Iterator] := ChangeRealEndianess(SecondDataBuffer[UI_Iterator]);
			END_FOR 
			//field specific data, keep separate at first. Then combine data into get struct in a later step.
			get.OutputField.ar_PowerlockCurrents[3][Phases.L1] := DataBuffer[0];
			get.OutputField.ar_PowerlockCurrents[3][Phases.L2] := DataBuffer[1];
			get.OutputField.ar_PowerlockCurrents[3][Phases.L3] := DataBuffer[2];
			get.OutputField.ar_PowerlockCurrents[3][Phases.N] := DataBuffer[3];

			ast_OutputPowerLockData[3].r_ActivePhasePower[phases.L1] := DataBuffer[4];
 	  		ast_OutputPowerLockData[3].r_ActivePhasePower[phases.L2] := DataBuffer[5];
			ast_OutputPowerLockData[3].r_ActivePhasePower[phases.L3] := DataBuffer[6];
			ast_OutputPowerLockData[3].r_ActivePhasePower[phases.AVG] := (DataBuffer[4] + DataBuffer[5] + DataBuffer[6])/3;
		                            
			ast_OutputPowerLockData[3].r_ApparentPhasePower[phases.L1] := DataBuffer[8];
	   		ast_OutputPowerLockData[3].r_ApparentPhasePower[phases.L2] := DataBuffer[9];
			ast_OutputPowerLockData[3].r_ApparentPhasePower[phases.L3] := DataBuffer[10];
			ast_OutputPowerLockData[3].r_ApparentPhasePower[phases.AVG] := (DataBuffer[8] + DataBuffer[9] + DataBuffer[10])/3;
		                            
			ast_OutputPowerLockData[3].r_ReactivePhasePower[phases.L1] := DataBuffer[12];
 	 		ast_OutputPowerLockData[3].r_ReactivePhasePower[phases.L2] := DataBuffer[13];
			ast_OutputPowerLockData[3].r_ReactivePhasePower[phases.L3] := DataBuffer[14];
			ast_OutputPowerLockData[3].r_ReactivePhasePower[phases.AVG] := (DataBuffer[12] + DataBuffer[13] + DataBuffer[14])/3;
		    				                        
			ast_OutputPowerLockData[3].r_ActivePower := DataBuffer[7];
			ast_OutputPowerLockData[3].r_ApparentPower := DataBuffer[11];
			ast_OutputPowerLockData[3].r_ReactivePower := DataBuffer[15];
									
			ast_OutputPowerLockData[3].ar_PowerFactor[Phases.L1] := DataBuffer[16];
			ast_OutputPowerLockData[3].ar_PowerFactor[Phases.L2] := DataBuffer[17];
			ast_OutputPowerLockData[3].ar_PowerFactor[Phases.L3] := DataBuffer[18];
			ast_OutputPowerLockData[3].ar_PowerFactor[Phases.AVG] := (DataBuffer[16] + DataBuffer[17] + DataBuffer[18])/3;
									
			ast_OutputPowerLockData[3].r_EnergyConsumed	:=  DataBuffer[26];
			ast_OutputPowerLockData[3].r_EnergySupplied 	:=	DataBuffer[30];
									
			ast_OutputPowerLockData[3].ar_THD[Phases.L1] := DataBuffer[47];
			ast_OutputPowerLockData[3].ar_THD[Phases.L2] := DataBuffer[48];
			ast_OutputPowerLockData[3].ar_THD[Phases.L3] := DataBuffer[49];
				
			ui_MBRetryCount := 0;
			sfctip := TRUE;
		ELSE
			ui_MBRetryCount := ui_MBRetryCount + 1;

			IF ui_MBRetryCount > 1 THEN
				get.events.b_MBCommWarning := TRUE;
			END_IF	
			
			//if comm fails 5 times in a row. try next input
			IF ui_MBRetryCount > 4 THEN
				get.Events.b_MBCommError := TRUE;
				sfctip := TRUE;
			END_IF
		END_IF
	END_IF
END_IF
END_ACTION

METHOD ChangeRealEndianess : REAL
VAR_INPUT
	InputReal	:	REAL;
END_VAR

VAR
	TestWord	:	WORD;
	TestByte	: ARRAY[0..3] OF BYTE;
END_VAR

MEMCPY(ADR(ChangeRealEndianess)+2, 	ADR(InputReal), 	2);
MEMCPY(ADR(ChangeRealEndianess), 	ADR(InputReal)+2, 	2);

memcpy(ADR(TestWord), ADR(InputReal), 2);
IF ((TestWord AND 2#0111111110000000) = 2#0111111110000000) THEN
	ChangeRealEndianess := 0;
END_IF
END_METHOD

ACTION ReadDataSFC:
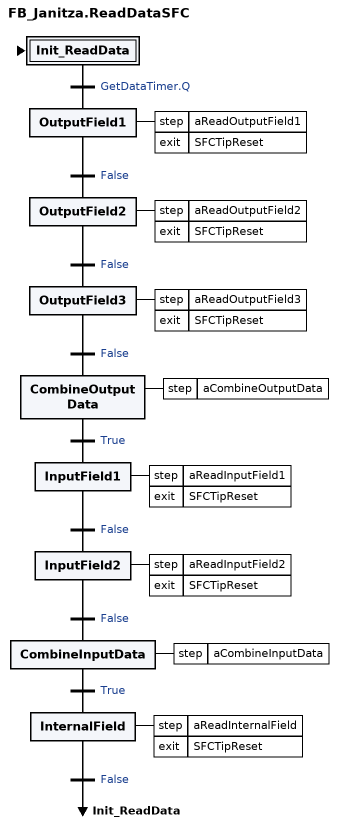
INITIAL_STEP Init_ReadData:
END_STEP
TRANSITION FROM Init_ReadData TO OutputField1
    := GetDataTimer.Q;
END_TRANSITION
STEP OutputField1:
    aReadOutputField1(N);  // step action
    SFCTipReset(P0);  // exit action
END_STEP
TRANSITION FROM OutputField1 TO OutputField2
    := False;
END_TRANSITION
STEP OutputField2:
    aReadOutputField2(N);  // step action
    SFCTipReset(P0);  // exit action
END_STEP
TRANSITION FROM OutputField2 TO OutputField3
    := False;
END_TRANSITION
STEP OutputField3:
    aReadOutputField3(N);  // step action
    SFCTipReset(P0);  // exit action
END_STEP
TRANSITION FROM OutputField3 TO CombineOutputData
    := False;
END_TRANSITION
STEP CombineOutputData:
    aCombineOutputData(N);  // step action
END_STEP
TRANSITION FROM CombineOutputData TO InputField1
    := True;
END_TRANSITION
STEP InputField1:
    aReadInputField1(N);  // step action
    SFCTipReset(P0);  // exit action
END_STEP
TRANSITION FROM InputField1 TO InputField2
    := False;
END_TRANSITION
STEP InputField2:
    aReadInputField2(N);  // step action
    SFCTipReset(P0);  // exit action
END_STEP
TRANSITION FROM InputField2 TO CombineInputData
    := False;
END_TRANSITION
STEP CombineInputData:
    aCombineInputData(N);  // step action
END_STEP
TRANSITION FROM CombineInputData TO InternalField
    := True;
END_TRANSITION
STEP InternalField:
    aReadInternalField(N);  // step action
    SFCTipReset(P0);  // exit action
END_STEP
TRANSITION FROM InternalField TO Init_ReadData
    := False;
END_TRANSITION
END_ACTION

ACTION SFCTipReset:
SFCTip := FALSE;
END_ACTION

END_FUNCTION_BLOCK

(* stored: Version 1.1.0.1, ProductVersion 3.1.4024.12
   POU FB_Janitza: Id {d3439d1b-beb1-49ad-8771-ebd77ff65768}, SpecialFunc None
   Folder SFC: Id {7b546ac8-05b5-4879-b9ec-fda86df5f1f4}
   Action aCombineInputData: Id {180e600d-b54b-4a85-85a4-80b021480939}
   Action aCombineOutputData: Id {e60d4201-2e5a-4e45-91b9-0987642fe282}
   Action aReadInputField1: Id {09026925-47af-4f0d-b345-026e75e997e6}
   Action aReadInputField2: Id {879d4ce2-fa80-469d-ae98-e3a65a92c6ac}
   Action aReadInternalField: Id {d526bcb8-a602-4936-a0ca-348cc77ced31}
   Action aReadOutputField1: Id {2560e15b-336a-4bdd-a5e9-c733f2196bcb}
   Action aReadOutputField2: Id {23a7dd3d-a6cf-41c7-9f6e-8f42bd580130}
   Action aReadOutputField3: Id {a2de4e77-9600-45d8-8e1d-937b9ee1205f}
   Method ChangeRealEndianess: Id {8c481591-1a82-403f-8748-c7bd77550c00}
   Action ReadDataSFC: Id {d47c650b-b078-4699-aabe-71eb457c26b2}
   Action SFCTipReset: Id {097b2a57-11df-4388-96f3-9b159a6b302d} *)
